// TwinCAT 3 PLC project Prozessmodell
// ProgramVersion: 3.1.4026.10
// libraries:
//   Tc2_Standard, * (Beckhoff Automation GmbH)
//   Tc2_System, * (Beckhoff Automation GmbH)
// project tree:
//   DUTs/ ObjectMode.TcDUT (not stored), ObjectState.TcDUT (not stored), SkillState.TcDUT (not stored), SystemState.TcDUT (not stored)
//   / PlcTask.TcTTO
//   POUs/01_Versuch_1/01_Skills/ SkillBasisGeruest.TcPOU (not stored), SkillNeu.TcPOU (not stored), TestSkill.TcPOU
//   POUs/01_Versuch_1/02_Skillprozess/ Skill_1.TcPOU
//   POUs/01_Versuch_1/03_Sequenz/ Sequenz_1.TcPOU
//   POUs/01_Versuch_1/ Arbeitsplan.TcPOU, Instanziierne.TcPOU (not stored)
//   POUs/02_Versuch_2/ BasisSkill.TcPOU, Instanziierung.TcPOU, TestSkill_1.TcPOU
//   POUs/ MAIN.TcPOU
// real-time tasks:
//   TASK PlcTask: cycle T#10ms, priority 20, ADS port 350
//   TASK PlcTask1: cycle T#10ms, priority 21, ADS port 351

CONFIGURATION Prozessmodell
    RESOURCE PLC ON TwinCAT3
        TASK PlcTask(INTERVAL := T#10ms, PRIORITY := 21);
        PROGRAM MAIN WITH PlcTask : MAIN;
    END_RESOURCE
END_CONFIGURATION

// ---- POUs/MAIN.TcPOU
PROGRAM MAIN
VAR
END_VAR

Instanziierung();

END_PROGRAM

// ---- POUs/02_Versuch_2/Instanziierung.TcPOU
PROGRAM Instanziierung
VAR
	Skill		:BasisSkill;
	TestSkill	:TestSkill_1;
END_VAR

Skill(); // BasisSkill
TestSkill(); // TestSkill_1

END_PROGRAM

// ---- POUs/02_Versuch_2/BasisSkill.TcPOU
FUNCTION_BLOCK BasisSkill
VAR_INPUT
	bExecute			:BOOL;				// Trigger für Ausführung von Skill
	bReset				:BOOL;				// Trigger für Reset von Skill
	iObjState			:ObjectState;		// Information über Zustand von Objekt
	iSysState			:SystemState;		// Information über Zustand von System
END_VAR
VAR_OUTPUT
	iMode				:ObjectMode;		// Steuerungsvariable für Anlagenmodell
	bDone				:BOOL;				// Information ob Skill ausgfeührt wurde
	bBusy				:BOOL;				// Information ob Skill im Moment ausgeführt wird
	bLimit				:BOOL;				// Information ob Skill an einem Limit angekommen ist
	bError				:BOOL;				// Information ob sich Skill in Fehlerzustand befindet
	iErrorID			:INT;				// Information um welchen Fehler es sich handelt
END_VAR
VAR
	iState				:SkillState;		// Information über Zustand von Skill
	bTargetReached		:BOOL;				// Information ob Prozessziel erreicht wurde
	bLimitReached		:BOOL;				// Information ob Limit erreicht wurde
	
END_VAR

CASE iState OF 
	0: // BEREIT
			// DO
			IF bExecute THEN
					iMode := 1;										// Starten des Objektes 
			END_IF	
				
			// TRANSITION	
			IF iObjState = 2 THEN
					iState := 1;									// Objekt wurde gestartet
				END_IF
// _________________________________________________________________________________________________________________________

	1: // LAUFEND
			// DO
				bBusy := TRUE;										// Skill wird ausgeführt
				
				IF bTargetReached OR bLimitReached THEN				// Prüfen ob Prozessziel erreicht wurde
					iMode := 2;
				END_IF
				
			// TRANSITION 
				IF iObjState = 3 THEN								// Transition zu ABGESCHLOSSEN
					bBusy := FALSE;									// Skill wird nicht mehr ausgeführt
					iState := 2;									// Objekt ist fertig und wieder bereit
				END_IF
				
				IF iObjState = 4 AND bTargetReached THEN			// Transition zu ERREICHT
					bTargetReached := FALSE;						// Zurücksetzen von Information
					bBusy := FALSE;									// Skill wird nicht mehr ausgeführt
					iState := 3;
				END_IF
				
				IF iObjState = 4  AND bLimitReached THEN			// Transition zu LIMIT
					bLimitReached := FALSE;							// Zurücksetzen von Information
					bBusy := FALSE;									// Skill wird nicht mehr ausgeführt
					iState := 4;
				END_IF
				
				IF iSysState = 3 THEN								// Transition wenn System das Orbjekt stopps
 					bBusy := FALSE;									// Skill wird nicht mehr ausgeführt
					iState := 0;
				END_IF
				
// _________________________________________________________________________________________________________________________
			
	2: // ABGESCHLOSSEN
			// DO
				bDone := TRUE;										// Skill wurde erfolgreich ausgeführt
				
			//  TRANSITION
				IF bDone THEN
					bDone := FALSE;									// Zurücksetzen von Skill
					iMode := 3;										// Resetten von Objekt
					iState := 0;
				END_IF
// _________________________________________________________________________________________________________________________

	3: // ERREICHT		
			// DO 
				bDone := TRUE;										// Skill wurde erfolgreich ausgeführt
				
				IF bDone THEN
					bDone := FALSE;									// Zurücksetzen von Output-Variable
					iMode := 3;										// Resetten von Objekt
					iState := 0;
				END_IF
			
			// TRANSITION
// _________________________________________________________________________________________________________________________

	4: // LIMIT
			// DO 
				bLimit := TRUE;										// Limit wurde erreicht
		
			// TRANSITION
				IF bLimit THEN
					bLimit := FALSE;								// Zurücksetzen von Output-Variable
					iMode := 3;										// Resetten von Objekt 
					iState := 0;
				END_IF
// _________________________________________________________________________________________________________________________

	5: // FEHLER
	
END_CASE

PROPERTY P_Runtime : TIME
GET
END_GET
END_PROPERTY

PROPERTY P_State : INT
GET
P_State := iState;
END_GET
END_PROPERTY

END_FUNCTION_BLOCK

// ---- POUs/01_Versuch_1/01_Skills/TestSkill.TcPOU
FUNCTION_BLOCK TestSkill
VAR_INPUT
	InVar_1			:BOOL;
	InVar_2			:BOOL;
END_VAR
VAR_OUTPUT
	OutVar_1		:BOOL;
END_VAR
VAR
END_VAR

END_FUNCTION_BLOCK

// ---- POUs/02_Versuch_2/TestSkill_1.TcPOU
FUNCTION_BLOCK TestSkill_1 EXTENDS BasisSkill
VAR_INPUT
END_VAR
VAR_OUTPUT
END_VAR
VAR
END_VAR

CASE iState OF 
	0: // BEREIT
			// DO
			IF bExecute THEN
					iMode := 1;										// Starten des Objektes 
			END_IF	
				
			// TRANSITION	
			IF iObjState = 2 THEN
					iState := 1;									// Objekt wurde gestartet
				END_IF
// _________________________________________________________________________________________________________________________

	1: // LAUFEND
			// DO
				bBusy := TRUE;										// Skill wird ausgeführt
				
				IF bTargetReached OR bLimitReached THEN				// Prüfen ob Prozessziel erreicht wurde
					iMode := 2;
				END_IF
				
			// TRANSITION 
				IF iObjState = 3 THEN								// Transition zu ABGESCHLOSSEN
					bBusy := FALSE;									// Skill wird nicht mehr ausgeführt
					iState := 2;									// Objekt ist fertig und wieder bereit
				END_IF
				
				IF iObjState = 4 AND bTargetReached THEN			// Transition zu ERREICHT
					bTargetReached := FALSE;						// Zurücksetzen von Information
					bBusy := FALSE;									// Skill wird nicht mehr ausgeführt
					iState := 3;
				END_IF
				
				IF iObjState = 4  AND bLimitReached THEN			// Transition zu LIMIT
					bLimitReached := FALSE;							// Zurücksetzen von Information
					bBusy := FALSE;									// Skill wird nicht mehr ausgeführt
					iState := 4;
				END_IF
				
				IF iSysState = 3 THEN								// Transition wenn System das Orbjekt stopps
 					bBusy := FALSE;									// Skill wird nicht mehr ausgeführt
					iState := 0;
				END_IF
				
// _________________________________________________________________________________________________________________________
			
	2: // ABGESCHLOSSEN
			// DO
				bDone := TRUE;										// Skill wurde erfolgreich ausgeführt
				
			//  TRANSITION
				IF bDone THEN
					bDone := FALSE;									// Zurücksetzen von Skill
					iMode := 3;										// Resetten von Objekt
					iState := 0;
				END_IF
// _________________________________________________________________________________________________________________________

	3: // ERREICHT		
			// DO 
				bDone := TRUE;										// Skill wurde erfolgreich ausgeführt
				
				IF bDone THEN
					bDone := FALSE;									// Zurücksetzen von Output-Variable
					iMode := 3;										// Resetten von Objekt
					iState := 0;
				END_IF
			
			// TRANSITION
// _________________________________________________________________________________________________________________________

	4: // LIMIT
			// DO 
				bLimit := TRUE;										// Limit wurde erreicht
		
			// TRANSITION
				IF bLimit THEN
					bLimit := FALSE;								// Zurücksetzen von Output-Variable
					iMode := 3;										// Resetten von Objekt 
					iState := 0;
				END_IF
// _________________________________________________________________________________________________________________________

	5: // FEHLER
	
END_CASE

END_FUNCTION_BLOCK

// ---- POUs/01_Versuch_1/02_Skillprozess/Skill_1.TcPOU
FUNCTION_BLOCK Skill_1
VAR_INPUT
	Var_1			:BOOL;
	Var_2			:BOOL;
END_VAR
VAR_OUTPUT
	
END_VAR
VAR
	Skill_1			:TestSkill;
END_VAR

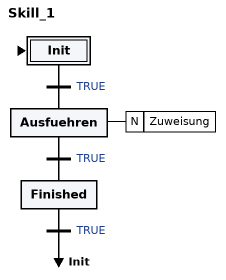
INITIAL_STEP Init:
END_STEP
TRANSITION FROM Init TO Ausfuehren
    := TRUE;
END_TRANSITION
STEP Ausfuehren:
    Zuweisung(N);
END_STEP
TRANSITION FROM Ausfuehren TO Finished
    := TRUE;
END_TRANSITION
STEP Finished:
END_STEP
TRANSITION FROM Finished TO Init
    := TRUE;
END_TRANSITION

ACTION Zuweisung:
Skill_1(InVar_1 := Var_1, InVar_2 := Var_2); // TestSkill
END_ACTION

END_FUNCTION_BLOCK

// ---- POUs/01_Versuch_1/03_Sequenz/Sequenz_1.TcPOU
FUNCTION_BLOCK Sequenz_1
VAR_INPUT
	Var_1		:BOOL;
	Var_2		:BOOL;
END_VAR
VAR_OUTPUT
	
END_VAR
VAR
	Skill_1			:TestSkill;
END_VAR

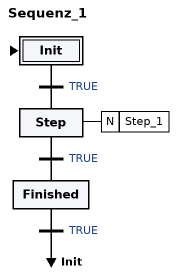
INITIAL_STEP Init:
END_STEP
TRANSITION FROM Init TO Step
    := TRUE;
END_TRANSITION
STEP Step:
    Step_1(N);
END_STEP
TRANSITION FROM Step TO Finished
    := TRUE;
END_TRANSITION
STEP Finished:
END_STEP
TRANSITION FROM Finished TO Init
    := TRUE;
END_TRANSITION

ACTION Step_1:
Skill_1(InVar_1 := Var_1, InVar_2 := Var_2); // TestSkill
END_ACTION

END_FUNCTION_BLOCK

// ---- POUs/01_Versuch_1/Arbeitsplan.TcPOU
PROGRAM Arbeitsplan
VAR
	Schritt_1		:Skill_1;
	Schritt_2		:Sequenz_1;
	
	Check			:BOOL;
	
	Var_1			:BOOL;
	Var_2			:BOOL;
	Var_3			:BOOL;
	Var_4			:BOOL;
END_VAR

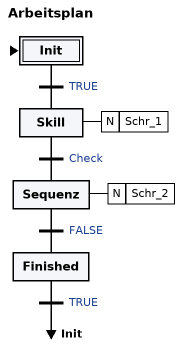
INITIAL_STEP Init:
END_STEP
TRANSITION FROM Init TO Skill
    := TRUE;
END_TRANSITION
STEP Skill:
    Schr_1(N);
END_STEP
TRANSITION FROM Skill TO Sequenz
    := Check;
END_TRANSITION
STEP Sequenz:
    Schr_2(N);
END_STEP
TRANSITION FROM Sequenz TO Finished
    := FALSE;
END_TRANSITION
STEP Finished:
END_STEP
TRANSITION FROM Finished TO Init
    := TRUE;
END_TRANSITION

ACTION Schr_1:
Schritt_1(Var_1 := Var_1, Var_2 := Var_2); // Skill_1
END_ACTION

ACTION Schr_2:
Schritt_2(Var_1 := Var_3, Var_2 := Var_4); // Sequenz_1
END_ACTION

END_PROGRAM
